PROGRAM MAIN
VAR
	bBool	: BOOL;
	iInt	: INT;
	
	fbGetEndTime: FB_GetEndTime;
	
	bTestTimeCalc	: BOOL;
	strEndTimeString	: STRING(255);
	strStartTimeString	: STRING(255);
END_VAR

iInt	:= iInt + 1;
IF(iInt > 100) THEN
	bBool	:= NOT(bBool); 
	iInt	:= 0;
END_IF

fbGetEndTime();
IF(bTestTimeCalc)THEN
	strEndTimeString	:= fbGetEndTime.GetEndTimeString(3900);
	bTestTimeCalc	:= FALSE;
END_IF

END_PROGRAM

(* stored: Version 1.1.0.1, ProductVersion 3.1.4024.12
   POU MAIN: Id {fbe2084b-4d56-4f1b-8424-b1f80ccbd60b}, SpecialFunc None *)
